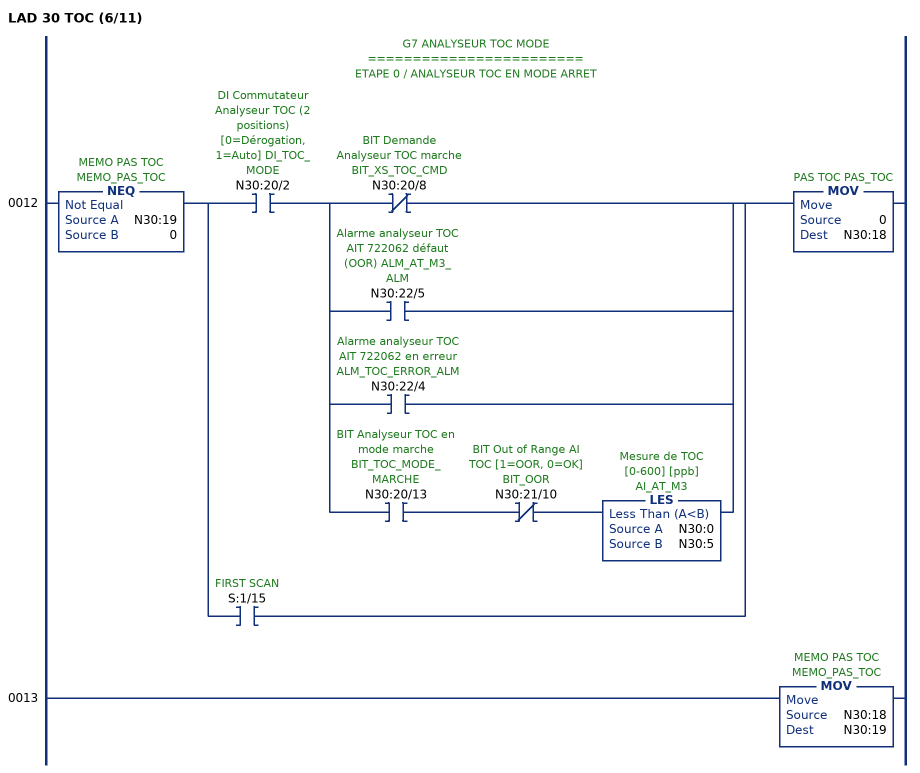
% Rung: 12 %
% G7 ANALYSEUR TOC MODE
% ========================
% ETAPE 0 / ANALYSEUR TOC EN MODE ARRET %
SOR NEQ N30:19 0 BST XIC N30:20/2 BST XIO N30:20/8 NXB XIC N30:22/5 NXB XIC N30:22/4 NXB XIC N30:20/13 XIO N30:21/10 LES N30:0 N30:5 BND NXB XIC S:1/15 BND MOV 0 N30:18 EOR
%   N30:19  MEMO_PAS_TOC  "MEMO PAS TOC" %
%   N30:20/2  DI_TOC_MODE  "DI Commutateur Analyseur TOC (2 positions) [0=Dérogation, 1=Auto]" %
%   N30:20/8  BIT_XS_TOC_CMD  "BIT Demande Analyseur TOC marche" %
%   N30:22/5  ALM_AT_M3_ALM  "Alarme analyseur TOC AIT 722062 défaut (OOR)" %
%   N30:22/4  ALM_TOC_ERROR_ALM  "Alarme analyseur TOC AIT 722062 en erreur" %
%   N30:20/13  BIT_TOC_MODE_MARCHE  "BIT Analyseur TOC en mode marche" %
%   N30:21/10  BIT_OOR  "BIT Out of Range AI TOC [1=OOR, 0=OK]" %
%   N30:0  AI_AT_M3  "Mesure de TOC [0-600] [ppb]" %
%   N30:5  AI_AT_M3_MIN  "Param05 TOC: Seuil d'initialisation de mesure de TOC [0-600] [ppb] <<4ppb>>" %
%   S:1/15  "FIRST SCAN" %
%   N30:18  PAS_TOC  "PAS TOC" %
% Rung: 13 %
SOR MOV N30:18 N30:19 EOR
%   N30:18  PAS_TOC  "PAS TOC" %
%   N30:19  MEMO_PAS_TOC  "MEMO PAS TOC" %

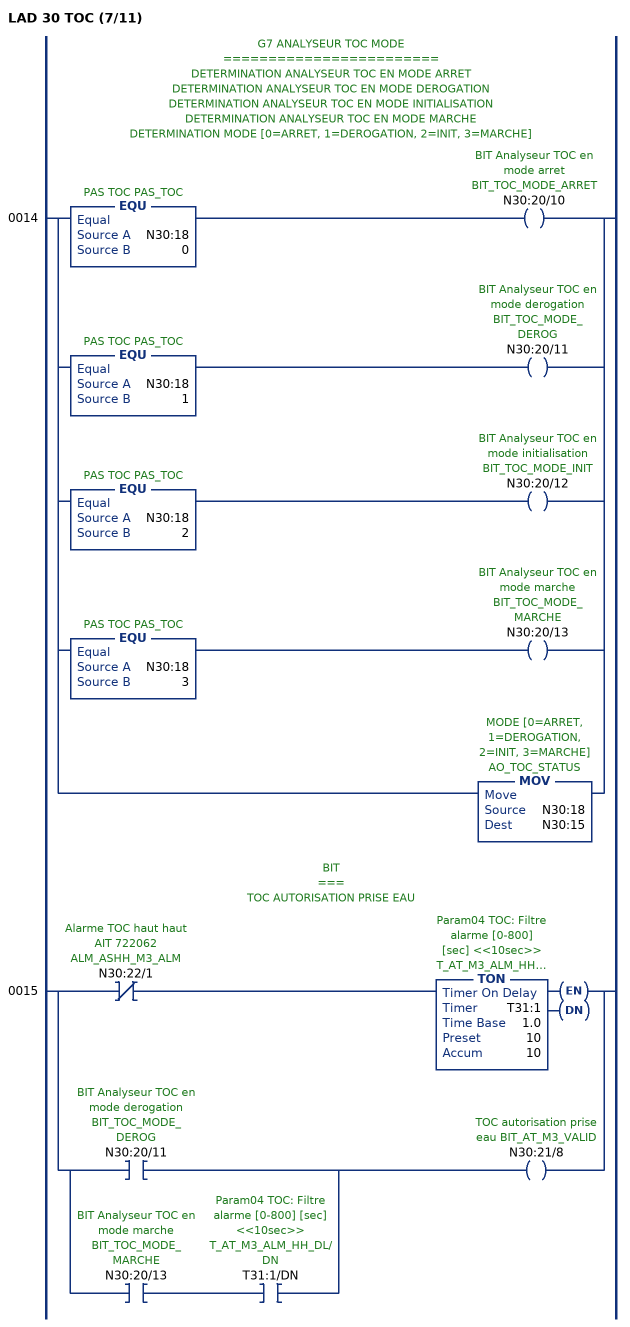
% Rung: 14 %
% G7 ANALYSEUR TOC MODE
% ========================
% DETERMINATION ANALYSEUR TOC EN MODE ARRET
% DETERMINATION ANALYSEUR TOC EN MODE DEROGATION
% DETERMINATION ANALYSEUR TOC EN MODE INITIALISATION
% DETERMINATION ANALYSEUR TOC EN MODE MARCHE
% DETERMINATION MODE [0=ARRET, 1=DEROGATION, 2=INIT, 3=MARCHE] %
SOR BST EQU N30:18 0 OTE N30:20/10 NXB EQU N30:18 1 OTE N30:20/11 NXB EQU N30:18 2 OTE N30:20/12 NXB EQU N30:18 3 OTE N30:20/13 NXB MOV N30:18 N30:15 BND EOR
%   N30:18  PAS_TOC  "PAS TOC" %
%   N30:20/10  BIT_TOC_MODE_ARRET  "BIT Analyseur TOC en mode arret" %
%   N30:20/11  BIT_TOC_MODE_DEROG  "BIT Analyseur TOC en mode derogation" %
%   N30:20/12  BIT_TOC_MODE_INIT  "BIT Analyseur TOC en mode initialisation" %
%   N30:20/13  BIT_TOC_MODE_MARCHE  "BIT Analyseur TOC en mode marche" %
%   N30:15  AO_TOC_STATUS  "MODE [0=ARRET, 1=DEROGATION, 2=INIT, 3=MARCHE]" %
% Rung: 15 %
% BIT
% ===
% TOC AUTORISATION PRISE EAU %
SOR BST XIO N30:22/1 TON T31:1 1.0 10 10 NXB BST XIC N30:20/11 NXB XIC N30:20/13 XIC T31:1/DN BND OTE N30:21/8 BND EOR
%   N30:22/1  ALM_ASHH_M3_ALM  "Alarme TOC haut haut AIT 722062" %
%   T31:1  T_AT_M3_ALM_HH_DL  "Param04 TOC: Filtre alarme [0-800] [sec] <<10sec>>" %
%   N30:20/11  BIT_TOC_MODE_DEROG  "BIT Analyseur TOC en mode derogation" %
%   N30:20/13  BIT_TOC_MODE_MARCHE  "BIT Analyseur TOC en mode marche" %
%   N30:21/8  BIT_AT_M3_VALID  "TOC autorisation prise eau" %

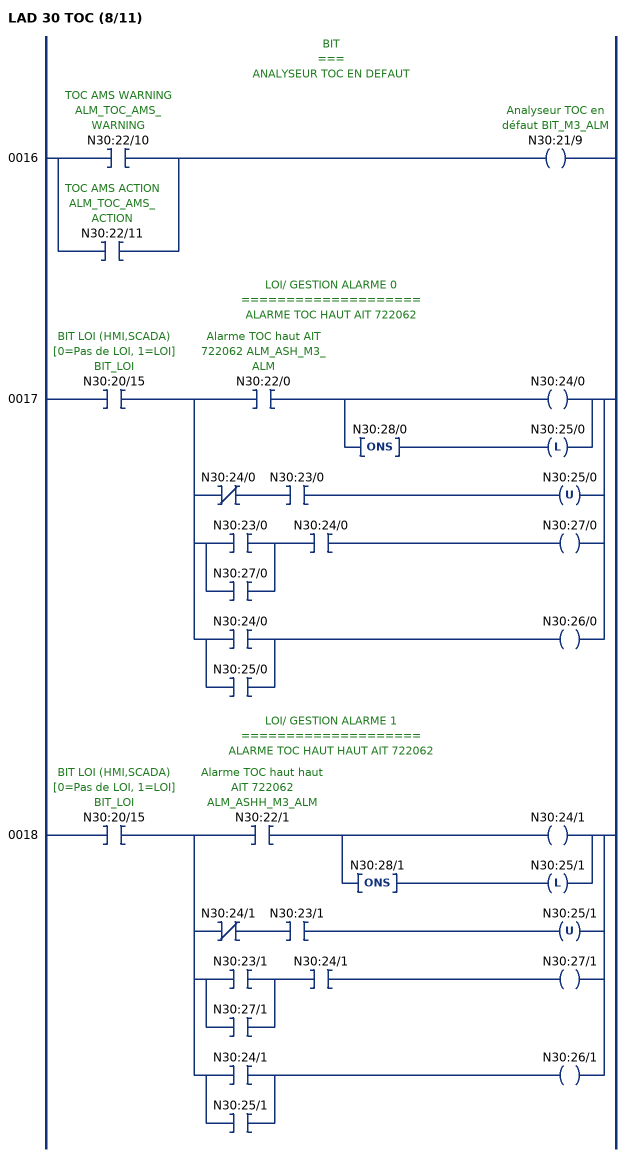
% Rung: 16 %
% BIT
% ===
% ANALYSEUR TOC EN DEFAUT %
SOR BST XIC N30:22/10 NXB XIC N30:22/11 BND OTE N30:21/9 EOR
%   N30:22/10  ALM_TOC_AMS_WARNING  "TOC AMS WARNING" %
%   N30:22/11  ALM_TOC_AMS_ACTION  "TOC AMS ACTION" %
%   N30:21/9  BIT_M3_ALM  "Analyseur TOC en défaut" %
% Rung: 17 %
% LOI/ GESTION ALARME 0
% ====================
% ALARME TOC HAUT AIT 722062 %
SOR XIC N30:20/15 BST XIC N30:22/0 BST OTE N30:24/0 NXB OSR N30:28/0 OTL N30:25/0 BND NXB XIO N30:24/0 XIC N30:23/0 OTU N30:25/0 NXB BST XIC N30:23/0 NXB XIC N30:27/0 BND XIC N30:24/0 OTE N30:27/0 NXB BST XIC N30:24/0 NXB XIC N30:25/0 BND OTE N30:26/0 BND EOR
%   N30:20/15  BIT_LOI  "BIT LOI (HMI,SCADA) [0=Pas de LOI, 1=LOI]" %
%   N30:22/0  ALM_ASH_M3_ALM  "Alarme TOC haut AIT 722062" %
% Rung: 18 %
% LOI/ GESTION ALARME 1
% ====================
% ALARME TOC HAUT HAUT AIT 722062 %
SOR XIC N30:20/15 BST XIC N30:22/1 BST OTE N30:24/1 NXB OSR N30:28/1 OTL N30:25/1 BND NXB XIO N30:24/1 XIC N30:23/1 OTU N30:25/1 NXB BST XIC N30:23/1 NXB XIC N30:27/1 BND XIC N30:24/1 OTE N30:27/1 NXB BST XIC N30:24/1 NXB XIC N30:25/1 BND OTE N30:26/1 BND EOR
%   N30:20/15  BIT_LOI  "BIT LOI (HMI,SCADA) [0=Pas de LOI, 1=LOI]" %
%   N30:22/1  ALM_ASHH_M3_ALM  "Alarme TOC haut haut AIT 722062" %

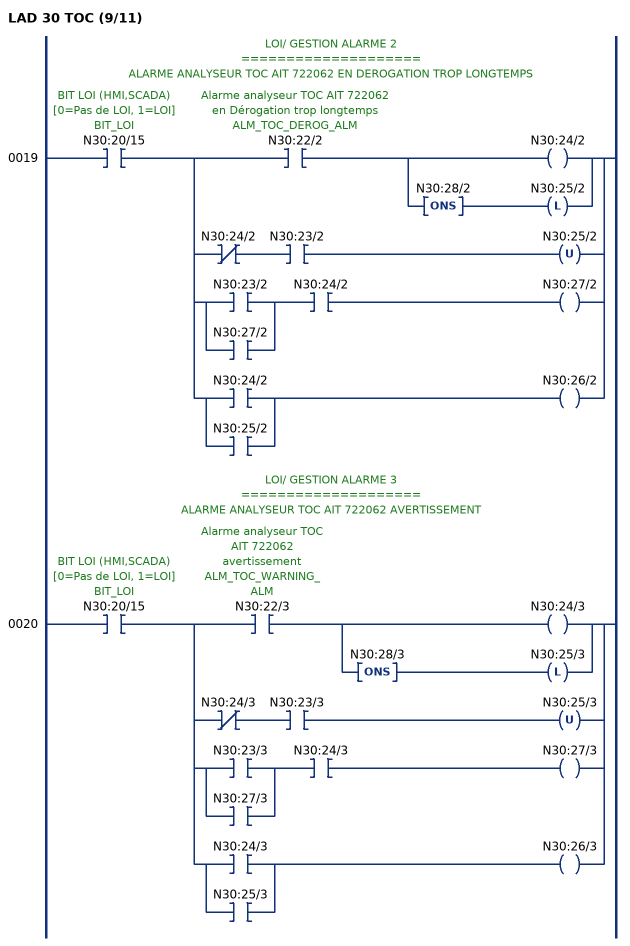
% Rung: 19 %
% LOI/ GESTION ALARME 2
% ====================
% ALARME ANALYSEUR TOC AIT 722062 EN DEROGATION TROP LONGTEMPS %
SOR XIC N30:20/15 BST XIC N30:22/2 BST OTE N30:24/2 NXB OSR N30:28/2 OTL N30:25/2 BND NXB XIO N30:24/2 XIC N30:23/2 OTU N30:25/2 NXB BST XIC N30:23/2 NXB XIC N30:27/2 BND XIC N30:24/2 OTE N30:27/2 NXB BST XIC N30:24/2 NXB XIC N30:25/2 BND OTE N30:26/2 BND EOR
%   N30:20/15  BIT_LOI  "BIT LOI (HMI,SCADA) [0=Pas de LOI, 1=LOI]" %
%   N30:22/2  ALM_TOC_DEROG_ALM  "Alarme analyseur TOC AIT 722062 en Dérogation trop longtemps" %
% Rung: 20 %
% LOI/ GESTION ALARME 3
% ====================
% ALARME ANALYSEUR TOC AIT 722062 AVERTISSEMENT %
SOR XIC N30:20/15 BST XIC N30:22/3 BST OTE N30:24/3 NXB OSR N30:28/3 OTL N30:25/3 BND NXB XIO N30:24/3 XIC N30:23/3 OTU N30:25/3 NXB BST XIC N30:23/3 NXB XIC N30:27/3 BND XIC N30:24/3 OTE N30:27/3 NXB BST XIC N30:24/3 NXB XIC N30:25/3 BND OTE N30:26/3 BND EOR
%   N30:20/15  BIT_LOI  "BIT LOI (HMI,SCADA) [0=Pas de LOI, 1=LOI]" %
%   N30:22/3  ALM_TOC_WARNING_ALM  "Alarme analyseur TOC AIT 722062 avertissement" %

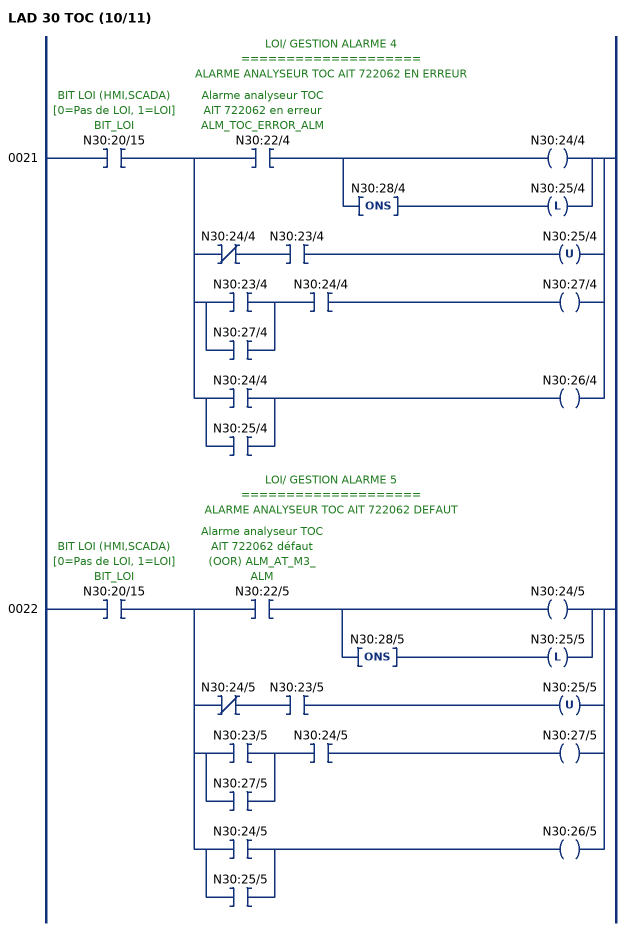
% Rung: 21 %
% LOI/ GESTION ALARME 4
% ====================
% ALARME ANALYSEUR TOC AIT 722062 EN ERREUR %
SOR XIC N30:20/15 BST XIC N30:22/4 BST OTE N30:24/4 NXB OSR N30:28/4 OTL N30:25/4 BND NXB XIO N30:24/4 XIC N30:23/4 OTU N30:25/4 NXB BST XIC N30:23/4 NXB XIC N30:27/4 BND XIC N30:24/4 OTE N30:27/4 NXB BST XIC N30:24/4 NXB XIC N30:25/4 BND OTE N30:26/4 BND EOR
%   N30:20/15  BIT_LOI  "BIT LOI (HMI,SCADA) [0=Pas de LOI, 1=LOI]" %
%   N30:22/4  ALM_TOC_ERROR_ALM  "Alarme analyseur TOC AIT 722062 en erreur" %
% Rung: 22 %
% LOI/ GESTION ALARME 5
% ====================
% ALARME ANALYSEUR TOC AIT 722062 DEFAUT %
SOR XIC N30:20/15 BST XIC N30:22/5 BST OTE N30:24/5 NXB OSR N30:28/5 OTL N30:25/5 BND NXB XIO N30:24/5 XIC N30:23/5 OTU N30:25/5 NXB BST XIC N30:23/5 NXB XIC N30:27/5 BND XIC N30:24/5 OTE N30:27/5 NXB BST XIC N30:24/5 NXB XIC N30:25/5 BND OTE N30:26/5 BND EOR
%   N30:20/15  BIT_LOI  "BIT LOI (HMI,SCADA) [0=Pas de LOI, 1=LOI]" %
%   N30:22/5  ALM_AT_M3_ALM  "Alarme analyseur TOC AIT 722062 défaut (OOR)" %

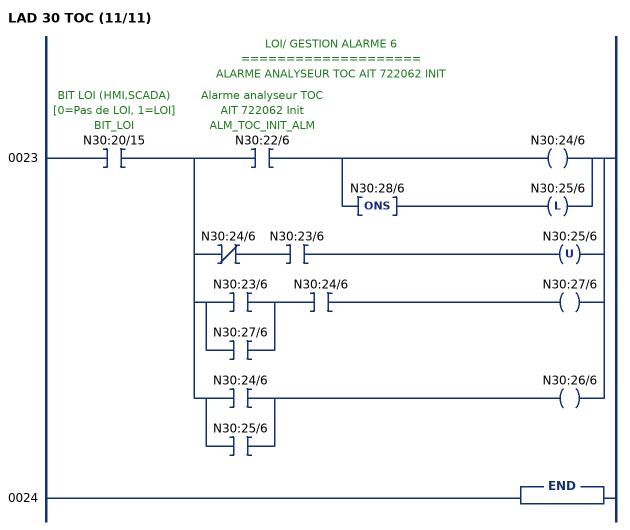
% Rung: 23 %
% LOI/ GESTION ALARME 6
% ====================
% ALARME ANALYSEUR TOC AIT 722062 INIT %
SOR XIC N30:20/15 BST XIC N30:22/6 BST OTE N30:24/6 NXB OSR N30:28/6 OTL N30:25/6 BND NXB XIO N30:24/6 XIC N30:23/6 OTU N30:25/6 NXB BST XIC N30:23/6 NXB XIC N30:27/6 BND XIC N30:24/6 OTE N30:27/6 NXB BST XIC N30:24/6 NXB XIC N30:25/6 BND OTE N30:26/6 BND EOR
%   N30:20/15  BIT_LOI  "BIT LOI (HMI,SCADA) [0=Pas de LOI, 1=LOI]" %
%   N30:22/6  ALM_TOC_INIT_ALM  "Alarme analyseur TOC AIT 722062 Init" %
% Rung: 24 %
SOR END EOR

OTHER DOCUMENTED ADDRESSES
  DFILE:30  "TOC Data Files/ Analyseu r TOC"
  DFILE:31  "TOC TIMER Data Files/ Analyseu r TOC"
  N7:10/3  "ALARM EMERGENCY STOP CIP"
  N30:10  A0_N30_10
  N30:13  A0_N30_13
  N30:14  A0_N30_14
  N30:16  A0_N30_16
  N30:17  A0_N30_17
  N30:20/3  DI_N30_20_3
  N30:20/4  DI_N30_20_4
  N30:20/5  DI_N30_20_5
  N30:20/6  DI_N30_20_6
  N30:20/7  DI_N30_20_7
  N30:20/9  BIT_TOC_MODE  "BIT Commutateur Analyseur TOC (2 positions) [0=Dérogation, 1=Auto]"
  N30:21/5  D0_N30_21_5
  N30:21/6  D0_N30_21_6
  N30:21/7  D0_N30_21_7
  N30:21/11  BIT_N30_21_11
  N30:21/12  BIT_N30_21_12
  N30:21/13  BIT_N30_21_13
  N30:21/14  BIT_N30_21_14
  N30:21/15  BIT_N30_21_15
  N30:22/7  ALM_N30_22_7
  N30:22/14  ALM_N30_22_14
  N30:22/15  ALM_N30_22_15
  N30:23  TOC_MOT_ACQ  "TOC GESTION ALARME/ MOT ACQUIT"
  N30:24  TOC_MOT_AL_EFF  "TOC GESTION ALARME/ MOT ALARME EFFECTIVE"
  N30:25  TOC_MOT_AL_NACQ  "TOC GESTION ALARME/ MOT ALARME NON ACQUITEE"
  N30:26  TOC_MOT_AL_EFF_NACQ  "TOC GESTION ALARME/ MOT ALARME EFFECTIVE NON ACQUITTEE"
  N30:27  TOC_MOT_AL_EFF_ACQ  "TOC GESTION ALARME/ MOT ALARME EFFECTIVE ACQUITTEE"
  N30:28  TOC_MOT_AL_F_M  "TOC GESTION ALARME/ MOT ALARME FRONT MONTANT"
  T4:38  "EPI-LOOP RETURN NOMINAL PRESSURE TEMPS X"
  T31:0/EN  "Param03 TOC: Temps max en mode Dérogation [0-720] [min] <<360min>>"
  T31:4/EN  T_TT_722011_LIMH_EN

REVISION NOTES
  93: Modification du seuil de démarrage deu distilateur N11:1
  94: Remplacement pile PLC 13/07/2007
  95: Ajout securite capot sur sprayball i6.9

DATA TABLE (non-zero values as saved)
DATA B3
% B3:0 % 0X0D00 0X11C1 0X0000 0X0000 0X0000 0X0000 0X0000 0X0000 0X0000 0X0000
DATA T4
% .PRE .ACC %
% T4:1 % 3 0
% T4:2 % 3 0
% T4:3 % 3 0
% T4:4 % 3 0
% T4:5 % 300 300
% T4:6 % 5 0
% T4:7 % 3 0
% T4:8 % 5 0
% T4:9 % 10 10
% T4:10 % 20 20
% T4:11 % 20 20
% T4:12 % 1 1
% T4:13 % 1 0
% T4:14 % 3 0
% T4:15 % 50 0
% T4:16 % 50 31
% T4:17 % 50 0
% T4:18 % 60 0
% T4:19 % 60 0
% T4:20 % 60 0
% T4:21 % 60 0
% T4:22 % 60 0
% T4:23 % 3 0
% T4:24 % 60 0
% T4:25 % 3 0
% T4:26 % 3 0
% T4:27 % 3 0
% T4:28 % 60 0
% T4:29 % 60 60
% T4:30 % 60 0
% T4:31 % 3600 0
% T4:32 % 3 0
% T4:33 % 5 0
% T4:34 % 3 3
% T4:35 % 3 0
% T4:36 % 3 0
% T4:37 % 300 300
% T4:38 % 10 0
% T4:40 % 3 3
% T4:41 % 3 3
% T4:54 % 3 3
% T4:58 % 3 0
DATA N7
% N7:10 % -32744
DATA B9
% B9:0 % 0X0000 0X0000 0X0000 0X0000 0X0004 0X1079 0X0050 0X8003 0X0050 0X0000
% B9:10 % 0X0050 0X07FF 0X0000 0X0000 0X0000 0X0000 0X0000 0X0000 0X0000 0X0000
DATA B10
% B10:0 % 0X0000 0X0000 0X0000 0XD5FA 0X0000 0X0280 0XFD80 0X0000 0X0000 0X0000
DATA N11
% N11:0 % 97 75 33 130 85 100 88 82 80 27
% N11:10 % 88 82 91 20 300 15 3 3 3 3
% N11:20 % 300 5 3 5 10 20 20 60 60 60
% N11:30 % 60 60 93 95 94 3 3 3 300 3
% N11:40 % 3 80 5 3600 0 600 3 1 1 50
% N11:50 % 50 3 3 -1 3 300 15 3 100 0
% N11:60 % 0 0 33 33 20 15 0 0 0 0
% N11:70 % 0 0 0 30 55
DATA N12
% N12:0 % 6242 15146 6242 0 0 0 0 0 0 0
DATA N13
% N13:0 % 4630 8713 11476 14205 11508 4042 8191 8191 4095 8191
% N13:10 % 6803 0
DATA N14
% N14:0 % 126 0 0 0 0 0 0 0 0 0
DATA N15
% N15:0 % 0 2 0 0 0 0 0 0 0 0
DATA N16
% N16:0 % 0 0 0 0 32765 32765
DATA N17
% N17:0 % 0 -53
DATA B18
% B18:0 % 0X0000 0X0700 0X7000 0X0000
DATA N19
% N19:0 % -16384 1 1 15 137 1 0 228 10 103
% N19:10 % 0 2 2304 0 -16384 2 1 15 137 2
% N19:20 % 0 164 10 103 0 2 2304 0 -31744 3
% N19:30 % 1 15 137 3 0 100 10 103 0 2
% N19:40 % 256 0 8192 4 1 15 137 5 0 32
% N19:50 % 0 0 0 2 3072 0 -16384 5 1 15
% N19:60 % 137 5 0 0 10 0 0 0 0 0
% N19:70 % -31744 6 1 15 137 6 0 0 10 0
% N19:80 % 0 0 0 0 -32768 3 1 15 137 6
% N19:90 % 0 100 10 56 0 2 4096 0
DATA T20
% .PRE .ACC %
% T20:1 % 300 0
% T20:2 % 15 0
% T20:4 % 5 0
% T20:11 % 300 0
% T20:12 % 15 0
% T20:14 % 3 0
% T20:21 % 300 0
% T20:22 % 15 0
% T20:24 % 3 0
DATA N24
% N24:0 % 15991 13107 7602 7537 10704 6554 10966 10442 10267 6816
% N24:10 % 10966 10442 15204 5898 94 13763 0 0 0 0
% N24:30 % 0 0 0 11578 11491 0 7646 0 3277 15073
% N24:40 % 11000 10267 0 0 0 5195 0 0 0 0
% N24:50 % 0 0 0 0 0 0 0 0 6554 0
% N24:60 % 0 0 0 8684 6554 5735 0 0 0 0
% N24:70 % 0 0 0 6144 11263
DATA N25
% N25:0 % 35 13180 93 1115 93 0 0 0 0 0
DATA N27
% N27:0 % -32727 0 10157 200 1 0 500 0 0 0
% N27:10 % 0 100 0 50 10287 -130 0 305 31520 2
% N27:20 % -32016 4605 10157 0 10287 0 0 0 0 0
% N27:30 % 0 0 10157 0 0 0 0 0 0 0
DATA N28
% N28:0 % -32223 0 6758 7 3 0 0 0 0 0
% N28:10 % 0 0 0 10 6887 -129 35 5886 -16194 1
% N28:20 % -20880 5251 6758 0 6886 5796
DATA N30
% N30:0 % 35 250 500 360 10 4 30 15 98 10
% N30:10 % 0 250 500 0 0 3 0 0 3 3
% N30:20 % 8455 263 0 0 0 0 0 0 0 0
DATA T31
% .PRE .ACC %
% T31:0 % 21600 0
% T31:1 % 10 10
% T31:2 % 1800 0
% T31:3 % 15 15
% T31:4 % 600 600
% T31:6 % 50 1
% T31:7 % 50 0
% T31:8 % 2 1
% T31:9 % 2 0
